{attribute 'qualified_only'}
{attribute 'strict'}
{attribute 'to_string'}
TYPE E_ModeCarrousel :
(
    INIT   := 0,
    AUTO   := 1,
    DEFAUT := 2
);
END_TYPE

(* stored: Version 1.1.0.1
   DUT E_ModeCarrousel: Id {c9c67771-c565-4939-bb9c-af675ead3ece} *)
